INTERFACE ITF_SaMController

METHOD Execute : BOOL
VAR_INPUT
	iNumberOfCommand		: INT;
END_VAR
END_METHOD

END_INTERFACE

(* stored: Version 1.1.0.1
   Itf ITF_SaMController: Id {c7f4a38b-e5fc-0e2c-38d0-203cc4e95405}
   Method Execute: Id {63ca3afc-c287-0bdd-12ae-e0974b7b3d54} *)
